(* CoDeSys 2.3 export: CALC_TRANSITIONS.EXP *)

(* POU lib/CALC_TRANSITIONS, FBD *)
FUNCTION_BLOCK CALC_TRANSITIONS
VAR_INPUT
	iSTATE										:	INT;
	xSTART									:	BOOL;
	xPROCESSING_PART					:	BOOL;
	xROTARY_STEP							:	BOOL;
	xPART_START_POS						:	BOOL;
	xPUNCH_PROXIMITY_SWITCH			:	BOOL;
	xPUNCH_FULLY_EXTENDED			:	BOOL;
	tPUNCH_DELAY							:	TIME;
	tPUNCH_FAIL_DELAY					:	TIME;
	xDRILL_PROXIMITY_SWITCH			:	BOOL;
	xDRILL_UPPER_LIMIT					:	BOOL;
	xDRILL_LOWER_LIMIT					:	BOOL;
	tDRILL_TIME								:	TIME;
	xPART_END_POS						:	BOOL;
END_VAR
VAR_OUTPUT
	_xT_0_1	:	BOOL;
	_xT_1_2	:	BOOL;
	_xT_2_3	:	BOOL;
	_xT_3_4	:	BOOL;
	_xT_4_5	:	BOOL;
	_xT_5_6	:	BOOL;
	_xT_6_7	:	BOOL;
	_xT_7_8	:	BOOL;
	_xT_8_0	:	BOOL;
END_VAR
VAR
	ton_punchDelay		:	TON;
	ton_punchFailDelay	:	TON;
	ton_drillTimer			:	TON;
	ft_partLeft				:	F_TRIG;
END_VAR
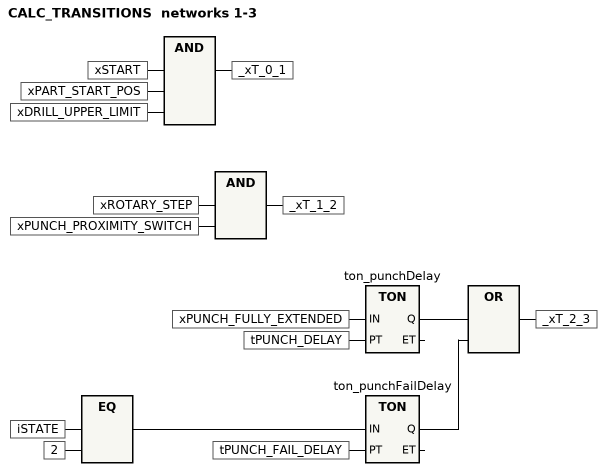
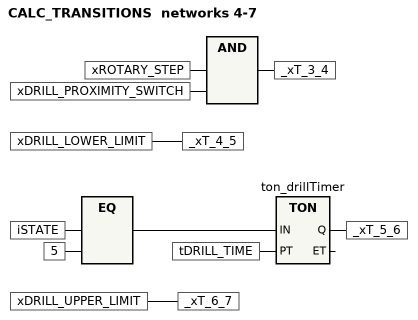
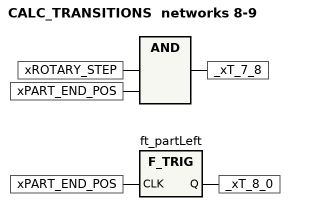
_FBD_ (* Function Block Diagram *)
NETWORK 1 start: (* The process may only start if a part is in the starting position, the drill is in its initial position and no other part is processing. *)
	AND(xSTART, xPART_START_POS, xDRILL_UPPER_LIMIT) => _xT_0_1
NETWORK 2 punchReached:
	AND(xROTARY_STEP, xPUNCH_PROXIMITY_SWITCH) => _xT_1_2
NETWORK 3 punchDone: (* Done if either the punch is fully extended or the part blocks the extension for a provided time. *)
	OR(ton_punchDelay:TON(IN: xPUNCH_FULLY_EXTENDED, PT: tPUNCH_DELAY), ton_punchFailDelay:TON(IN: EQ(iSTATE, 2), PT: tPUNCH_FAIL_DELAY)) => _xT_2_3
NETWORK 4 drillReached:
	AND(xROTARY_STEP, xDRILL_PROXIMITY_SWITCH) => _xT_3_4
NETWORK 5 drillLowered:
	xDRILL_LOWER_LIMIT => _xT_4_5
NETWORK 6 drillComplete:
	ton_drillTimer:TON(IN: EQ(iSTATE, 5), PT: tDRILL_TIME) => _xT_5_6
NETWORK 7 drillRaised:
	xDRILL_UPPER_LIMIT => _xT_6_7
NETWORK 8 endPosReached:
	AND(xROTARY_STEP, xPART_END_POS) => _xT_7_8
NETWORK 9 partLeft:
	ft_partLeft:F_TRIG(CLK: xPART_END_POS) => _xT_8_0
_END_FBD_
(* the same logic as Structured Text *)
(* Network 1: The process may only start if a part is in the starting position, the drill is in its initial position and no other part is processing. *)
start:
_xT_0_1 := xSTART AND xPART_START_POS AND xDRILL_UPPER_LIMIT;
(* Network 2 *)
punchReached:
_xT_1_2 := xROTARY_STEP AND xPUNCH_PROXIMITY_SWITCH;
(* Network 3: Done if either the punch is fully extended or the part blocks the extension for a provided time. *)
punchDone:
ton_punchDelay(IN := xPUNCH_FULLY_EXTENDED, PT := tPUNCH_DELAY);
ton_punchFailDelay(IN := iSTATE = 2, PT := tPUNCH_FAIL_DELAY);
_xT_2_3 := ton_punchDelay.Q OR ton_punchFailDelay.Q;
(* Network 4 *)
drillReached:
_xT_3_4 := xROTARY_STEP AND xDRILL_PROXIMITY_SWITCH;
(* Network 5 *)
drillLowered:
_xT_4_5 := xDRILL_LOWER_LIMIT;
(* Network 6 *)
drillComplete:
ton_drillTimer(IN := iSTATE = 5, PT := tDRILL_TIME);
_xT_5_6 := ton_drillTimer.Q;
(* Network 7 *)
drillRaised:
_xT_6_7 := xDRILL_UPPER_LIMIT;
(* Network 8 *)
endPosReached:
_xT_7_8 := xROTARY_STEP AND xPART_END_POS;
(* Network 9 *)
partLeft:
ft_partLeft(CLK := xPART_END_POS);
_xT_8_0 := ft_partLeft.Q;
END_FUNCTION_BLOCK
